// TIA Portal V17 export
// export: Created 2025-03-10T13:12:01.5910403Z, ExportSetting WithDefaults, DisplayName Totally Integrated Automation Portal, DisplayVersion V17 Update 8, DisplayName TIA Portal Openness, DisplayVersion V17 Update 8, DisplayName TIA Portal Version Control Interface, DisplayVersion V17, DisplayName SINAMICS Startdrive Advanced, DisplayVersion V17 SP2, DisplayName SINAMICS Startdrive G110M, G120, G120C, G120D, G120P, G115D, DisplayVersion V17 SP2, DisplayName SINAMICS Startdrive G130, G150, S120, S150, SINAMICS MV, S210, DisplayVersion V17 SP2, DisplayName STEP 7 Professional, DisplayVersion V17 Update 8, DisplayName SINUMERIK ONE STEP 7 Toolbox, DisplayVersion V17 Update 12, DisplayName SINUMERIK 840D sl STEP 7 Toolbox, DisplayVersion V17 Update 12, DisplayName STEP 7 Safety, DisplayVersion V17 Update 6, DisplayName WinCC Advanced, DisplayVersion V17 Update 8
TYPE "LBP_typePowerrideInput"
TITLE = Powerride image / Imagen de powerride / Powerride Abbild
// Input image of powerride / Imagen de entrada de powerride / Eingangsabbild von Powerride
// stored: IsFailsafeCompliant false
   STRUCT
      pushButton : Bool;   // TRUE, wenn Taster gedrückt / true, when push button pressed / TRUE, cuando el pulsador está accionado
      reserved01 : Bool;
      reserved02 : Bool;
      reserved03 : Bool;
      reserved04 : Bool;
      reserved05 : Bool;
      reserved06 : Bool;
      reserved07 : Bool;
      powerrideCounter : USInt;   // [0...255] Override-Schalterposition / [0..255] Override switch position / [0...255] Posición de interruptor en corrección
   END_STRUCT;
END_TYPE
